Fanuc KAREL source: kt00032.KL

-- PROVISIONAL review KL for V770-1; original PC SHA256 89c0a8350bb801f58b8e60f7f58d808bf467b92fb247d22275b907ede3b9d225
-- Incomplete behavior may be omitted. Consult companion uncertainty JSON. Do not deploy.
PROGRAM KT00032
%NOLOCKGROUP
VAR
  OUT : REAL
-- UNRESOLVED_DECL H1 type=002017
-- UNRESOLVED_DECL H2 type=002017
BEGIN
  -- UNRESOLVED_PC offsets 5-19; opcodes 2E,22,9D,33,B4
  -- UNRESOLVED_PC offsets 24-38; opcodes 2E,22,9D,33,B4
  -- UNRESOLVED_PC offsets 43-57; opcodes 2E,22,9D,33,B4
  -- UNRESOLVED_PC offsets 62-76; opcodes 2E,22,9D,33,B4
  -- UNRESOLVED_PC offsets 81-107; opcodes 22,9D,33,B3,22,9D,33,B3,52,64,23
  -- UNRESOLVED_PC offsets 112-116; opcodes 7F
END KT00032
